// TIA Portal V19 export
TYPE "PTrk_Item"
// stored: Access Published
   STRUCT
      P_ID : DInt;   // ID parte
      O_ID : DInt;   // ID ordine
      C_ID : DInt;   // ID rotolo
      Quality : Int;   // Qualità: UNKNOW;GOOD;BAD...
      Beam_Code : Int;   // Codice Pezzo: 0= SG formato da una singola parte; 1= C/S = Formato da due parti accoppiate
      PLen_Meas : Real;   // Lunghezza parte misurata (tra 2 tagli)
      W_A : Real;   // Dim. base (W) = Altezza in impilamento (A)
      H_B : Real;   // Dim. altezza (H) = base in impilamento (B)
      ShiftDone : Bool;   // Sfalsamento su A03 Pos.1 eseguito
   END_STRUCT;
END_TYPE
